FUNCTION_BLOCK OrderedDictionaryForwardEnumerator_TestSuite EXTENDS TcUnit.FB_TestSuite
VAR
END_VAR

CheckIsValidAtStart();
CheckMoveNextReturnsFalseAtTheEnd();
CheckMoveNextReturnsTrueSingleItem();
CheckMoveNextReturnsFalseWhenEmpty();
CheckMoveNextReturnsTrueMultipleItems();
CheckReset();
CheckTryGet();
CheckTryGetTo();
CheckWorksWithArrays();
CheckWorksWithIntegers();
CheckWorksWithStrings();

METHOD PRIVATE CheckIsValidAtStart
VAR
	result : BOOL;
	dictionary : OrderedDictionary;
	enumerator : I_ForwardEnumerator;
END_VAR
TEST('CheckIsValidAtStart');

enumerator := dictionary.GetEnumerator();

result := enumerator.IsValid;
enumerator.Dispose();

AssertTrue(
	Condition := result,
	Message := 'IsValid returned false'
);

TEST_FINISHED();
END_METHOD

METHOD PRIVATE CheckMoveNextReturnsFalseAtTheEnd
VAR
	in1 : INT := 123;
	result : BOOL;
	dictionary : OrderedDictionary;
	enumerator : I_ForwardEnumerator;
END_VAR
TEST('CheckMoveNextReturnsFalseAtTheEnd');

dictionary.TryAdd('a',in1);
enumerator := dictionary.GetEnumerator();

enumerator.MoveNext();
result := enumerator.MoveNext();

enumerator.Dispose();

AssertFalse(result,
    'MoveNext did not correctly signal the end of the enumeration');
	
TEST_FINISHED();
END_METHOD

METHOD PRIVATE CheckMoveNextReturnsFalseWhenEmpty
VAR
	result : BOOL;
	dictionary : OrderedDictionary;
	enumerator : I_ForwardEnumerator;
	count : DINT;
END_VAR
TEST('CheckMoveNextReturnsFalseWhenEmpty');

count := dictionary.Count;
enumerator := dictionary.GetEnumerator();

result := enumerator.MoveNext();
enumerator.Dispose();

AssertFalse(Condition := result,
    Message := 'MoveNext did not correctly signal the end of the enumeration');

TEST_FINISHED();
END_METHOD

METHOD PRIVATE CheckMoveNextReturnsTrueMultipleItems
VAR
	in1 : INT := 123;
	in2 : INT := 456;
	in3 : INT := 789;
	result : BOOL;
	dictionary : OrderedDictionary;
	enumerator : I_ForwardEnumerator;
END_VAR
TEST('CheckMoveNextReturnsTrueMultipleItems');

dictionary.TryAdd('a',in1);
dictionary.TryAdd('b',in2);
dictionary.TryAdd('c',in3);
enumerator := dictionary.GetEnumerator();

result := enumerator.MoveNext();
enumerator.Dispose();

AssertTrue(result, 'MoveNext did not correctly signal there were more items to follow');

TEST_FINISHED();
END_METHOD

METHOD PRIVATE CheckMoveNextReturnsTrueSingleItem
VAR
	in1 : INT := 123;
	result : BOOL;
	dictionary : OrderedDictionary;
	enumerator : I_ForwardEnumerator;
END_VAR
TEST('CheckMoveNextReturnsTrueSingleItem');

dictionary.TryAdd('a',in1);
enumerator := dictionary.GetEnumerator();

result := enumerator.MoveNext();
enumerator.Dispose();

AssertTrue(result,
    'MoveNext did not correctly signal there were more items to follow');
	
TEST_FINISHED();
END_METHOD

METHOD PRIVATE CheckReset
VAR
	in1 : ARRAY [0..1] OF REAL := [0.1,2.3];
	in2 : ARRAY [0..1] OF REAL := [1.2,3.4];
	in3 : ARRAY [0..1] OF REAL := [2.3,4.5];
	out : ARRAY [0..1] OF REAL;
	expected : ARRAY [0..1] OF REAL := [0.1,2.3];
	dictionary : OrderedDictionary;
	enumerator : I_ForwardEnumerator;
END_VAR
TEST('CheckReset');

dictionary.TryAdd('a',in1);
dictionary.TryAdd('b',in2);
dictionary.TryAdd('c',in3);

enumerator := dictionary.GetEnumerator();

enumerator.MoveNext();
enumerator.MoveNext();
enumerator.Reset();
enumerator.MoveNext();
enumerator.TryGet(out);

enumerator.Dispose();

AssertEquals(
	Expected := expected,
	Actual := out,
	Message := 'Did not produce the expected result'
);

TEST_FINISHED();
END_METHOD

METHOD PRIVATE CheckTryGet
VAR
	in : INT := 123;
	out : INT;
	expected : INT := 123;
	result : BOOL;
	dictionary : OrderedDictionary;
	enumerator : I_ForwardEnumerator;
END_VAR
TEST('CheckTryGet');

dictionary.TryAdd('a',in);
enumerator := dictionary.GetEnumerator();
enumerator.MoveNext();

result := enumerator.TryGet(out);
enumerator.Dispose();

AssertTrue(
	Condition := result,
	Message := 'Method returned false'
);

AssertEquals(
	Expected := expected,
	Actual := out,
	Message := 'Did not produce the expected result'
);

TEST_FINISHED();
END_METHOD

METHOD PRIVATE CheckTryGetTo
VAR
	in : INT := 123;
	out : INT;
	expected : INT := 123;
	result : BOOL;
	dictionary : OrderedDictionary;
	enumerator : I_ForwardEnumerator;
END_VAR
TEST('CheckTryGetTo');

dictionary.TryAdd('a',in);
enumerator := dictionary.GetEnumerator();
enumerator.MoveNext();

result := enumerator.TryGetTo(ADR(out),SIZEOF(out));
enumerator.Dispose();

AssertTrue(
	Condition := result,
	Message := 'Method returned false'
);

AssertEquals(
	Expected := expected,
	Actual := out,
	Message := 'Did not produce the expected result'
);

TEST_FINISHED();
END_METHOD

METHOD PRIVATE CheckWorksWithArrays
VAR
	in1 : ARRAY [0..1] OF REAL := [0.1,2.3];
	in2 : ARRAY [0..1] OF REAL := [1.2,3.4];
	in3 : ARRAY [0..1] OF REAL := [2.3,4.5];
	out1 : ARRAY [0..1] OF REAL;
	out2 : ARRAY [0..1] OF REAL;
	out3 : ARRAY [0..1] OF REAL;
	expected1 : ARRAY [0..1] OF REAL := [0.1,2.3];
	expected2 : ARRAY [0..1] OF REAL := [1.2,3.4];
	expected3 : ARRAY [0..1] OF REAL := [2.3,4.5];
	dictionary : OrderedDictionary;
	enumerator : I_ForwardEnumerator;
END_VAR
TEST('CheckWorksWithArrays');

dictionary.TryAdd('c',in1);
dictionary.TryAdd('b',in2);
dictionary.TryAdd('a',in3);

enumerator := dictionary.GetEnumerator();

enumerator.MoveNext();
enumerator.TryGet(out1);
enumerator.MoveNext();
enumerator.TryGet(out2);
enumerator.MoveNext();
enumerator.TryGet(out3);

enumerator.Dispose();

AssertEquals(
	Expected := expected1,
	Actual := out1,
	Message := 'Did not produce the expected 1st result'
);

AssertEquals(
	Expected := expected2,
	Actual := out2,
	Message := 'Did not produce the expected 2nd result'
);

AssertEquals(
	Expected := expected3,
	Actual := out3,
	Message := 'Did not produce the expected 3rd result'
);

TEST_FINISHED();
END_METHOD

METHOD PRIVATE CheckWorksWithIntegers
VAR
	in1 : INT := 123;
	in2 : INT := 234;
	in3 : INT := 345;
	out1 : INT;
	out2 : INT;
	out3 : INT;
	expected1 : INT := 123;
	expected2 : INT := 234;
	expected3 : INT := 345;
	dictionary : OrderedDictionary;
	enumerator : I_ForwardEnumerator;
END_VAR
TEST('CheckWorksWithIntegers');

dictionary.TryAdd('c',in1);
dictionary.TryAdd('b',in2);
dictionary.TryAdd('a',in3);

enumerator := dictionary.GetEnumerator();

enumerator.MoveNext();
enumerator.TryGet(out1);
enumerator.MoveNext();
enumerator.TryGet(out2);
enumerator.MoveNext();
enumerator.TryGet(out3);

enumerator.Dispose();

AssertEquals(
	Expected := expected1,
	Actual := out1,
	Message := 'Did not produce the expected 1st result'
);

AssertEquals(
	Expected := expected2,
	Actual := out2,
	Message := 'Did not produce the expected 2nd result'
);

AssertEquals(
	Expected := expected3,
	Actual := out3,
	Message := 'Did not produce the expected 3rd result'
);

TEST_FINISHED();
END_METHOD

METHOD PRIVATE CheckWorksWithStrings
VAR
	in1 : STRING := 'test1';
	in2 : STRING := 'test2';
	in3 : STRING := 'test3';
	out1 : STRING;
	out2 : STRING;
	out3 : STRING;
	expected1 : STRING := 'test1';
	expected2 : STRING := 'test2';
	expected3 : STRING := 'test3';
	dictionary : OrderedDictionary;
	enumerator : I_ForwardEnumerator;
END_VAR
TEST('CheckWorksWithStrings');

dictionary.TryAdd('c',in1);
dictionary.TryAdd('b',in2);
dictionary.TryAdd('a',in3);

enumerator := dictionary.GetEnumerator();

enumerator.MoveNext();
enumerator.TryGet(out1);
enumerator.MoveNext();
enumerator.TryGet(out2);
enumerator.MoveNext();
enumerator.TryGet(out3);

enumerator.Dispose();

AssertEquals(
	Expected := expected1,
	Actual := out1,
	Message := 'Did not produce the expected 1st result'
);

AssertEquals(
	Expected := expected2,
	Actual := out2,
	Message := 'Did not produce the expected 2nd result'
);

AssertEquals(
	Expected := expected3,
	Actual := out3,
	Message := 'Did not produce the expected 3rd result'
);

TEST_FINISHED();
END_METHOD

END_FUNCTION_BLOCK

(* stored: Version 1.1.0.1, ProductVersion 3.1.4024.12
   POU OrderedDictionaryForwardEnumerator_TestSuite: Id {50d3c1f1-8d28-4484-9f0d-4cf9ec5c3f1d}, SpecialFunc None
   Method CheckIsValidAtStart: Id {2afa093e-a8df-4358-baf2-eb4cc48a10bc}
   Method CheckMoveNextReturnsFalseAtTheEnd: Id {39f87f0a-adac-4108-a1cc-c186e15e6410}
   Method CheckMoveNextReturnsFalseWhenEmpty: Id {a756bd7b-32dc-4036-bcca-6ec1d266f1e3}
   Method CheckMoveNextReturnsTrueMultipleItems: Id {43a6bc39-42eb-4381-885d-4e727df7a798}
   Method CheckMoveNextReturnsTrueSingleItem: Id {dfd85771-ac9d-40e0-9c6b-df2d493c3c0c}
   Method CheckReset: Id {c852745a-56a5-42c4-bc2b-2364c32bcb05}
   Method CheckTryGet: Id {9a3c7ca8-96fd-43a9-bc2f-df4b692f7e01}
   Method CheckTryGetTo: Id {1e0b6213-4f90-47da-9017-f1194f125972}
   Method CheckWorksWithArrays: Id {8a342c84-adfe-4179-aecd-a753dd2ecdcd}
   Method CheckWorksWithIntegers: Id {25677e29-d9a6-412f-860b-eeae6d514dd7}
   Method CheckWorksWithStrings: Id {41446830-726d-4934-951f-37c8421ddcc8} *)
